KUKA KRL program: style1drop1opt1.src, style1drop1opt1.dat

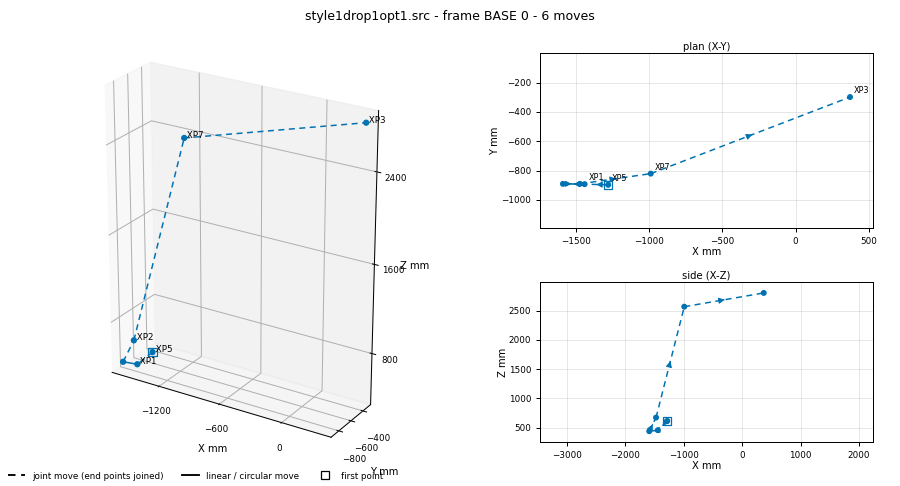
[picture p0: tool path of style1drop1opt1.src in frame BASE 0, 6 of 7 moves have a stored position in this frame; points joined in program order, loops and branches not executed]
--- style1drop1opt1.src ---
&ACCESS RVO1
&REL 222
&COMMENT 03-10-R1 DROP CONVEYOR
&PARAM EDITMASK = *
&PARAM DISKPATH = KRC:\R1\Program\StyleDrops\Options
DEF Style1Drop1Opt1( )
   ;FOLD INI
      ;FOLD BASISTECH INI
         GLOBAL INTERRUPT DECL 3 WHEN $STOPMESS==TRUE DO IR_STOPM ( )
         INTERRUPT ON 3
         BAS (#INITMOV,0 )
      ;ENDFOLD (BASISTECH INI)
      ;FOLD USER INI
         ;Make your modifications here

      ;ENDFOLD (USER INI)
   ;ENDFOLD (INI)
;********************************
; Gestamp Standards
; Line - BMW G65 (cell 03)
; Robot 03-10-R1 (BMW-03-10-R1-MH1)
; Application - DROP THE GOOD PART AT DROPOFF 1 (CONVEYOR)
;********************************
; CALLED BY Style1Opt1 WHEN BOTH NUT CHECKS PASSED. PLACES THE PART AT AtDrop3, OPENS
; GRIPPER 1, WAITS FOR THE GRIPPER EMPTY, LEAVES AND RETURNS HOME.
;NOTE: THE PART IN THE GRIPPER IS NOT CONFIRMED BEFORE OPENING (F40)
;DROPOFF 1 REQUEST - AC_DropOffCheck(1): WAIT SIGNAL $IN[75] di075DropOffMachine1 ON
;(WAITING MESSAGE, NO TIMEOUT), THEN SIGNALS $OUT[75] do075DropOffClear1 OFF,
;$OUT[25] do025DropClearTooling OFF
;WARNING: HIDDEN AC_CmdParam=2 - CONFIRMING THIS FORM REGENERATES AC_DropOffCheck(2) (F21)
;FOLD DropOff[1] Request
;FOLD ;%{h}
;Params IlfProvider=ac_zoneilf; AC_CmdZones=DropOff; AC_CmdParam=2; AC_ZoneRepo=False; AC_Blending=False
;ENDFOLD
AC_DropOffCheck (1)
;ENDFOLD

;APPROACH DROPOFF 1 - P5, P1, AtDrop3 (DROP POSITION)
;FOLD PTP P5 CONT Vel=100 % PDAT10 Tool[1]:TOOL 1 Base[0];%{PE}%R 8.3.43,%MKUKATPBASIS,%CMOVE,%VPTP,%P 1:PTP, 2:P5, 3:C_DIS, 5:100, 7:PDAT10
$BWDSTART=FALSE
PDAT_ACT=PPDAT10
FDAT_ACT=FP5
BAS(#PTP_PARAMS,100)
PTP XP5 C_DIS
;ENDFOLD
;FOLD PTP P1 Vel=100 % PDAT1 Tool[1]:TOOL 1 Base[0];%{PE}%R 8.3.43,%MKUKATPBASIS,%CMOVE,%VPTP,%P 1:PTP, 2:P1, 3:, 5:100, 7:PDAT1
$BWDSTART=FALSE
PDAT_ACT=PPDAT1
FDAT_ACT=FP1
BAS(#PTP_PARAMS,100)
PTP XP1
;ENDFOLD
;FOLD LIN AtDrop3 Vel=2 m/s CPDAT1 Tool[1]:TOOL 1 Base[0];%{PE}%R 8.3.43,%MKUKATPBASIS,%CMOVE,%VLIN,%P 1:LIN, 2:AtDrop3, 3:, 5:2, 7:CPDAT1
$BWDSTART=FALSE
LDAT_ACT=LCPDAT1
FDAT_ACT=FAtDrop3
BAS(#CP_PARAMS,2)
LIN XAtDrop3
;ENDFOLD

;GRIPPER 1 OPEN - SIGNALS $OUT[249] do249Group1Home ON, $OUT[250] do250Group1Work OFF, WAIT 0.2 S,
;THEN CHECK $IN[257] di257Cylinder1Home ON, $IN[258] di258Cylinder1Work OFF (STRATEGY 1)
;WARNING: THE HIDDEN FORM PARAMETERS SAY setgripper=4;setstate=2 - OPENING AND CONFIRMING THIS
;  FORM REGENERATES GRPg_SetStateAndCheck(4, 2, ...), AN INACTIVE GRIPPER: NOTHING OPENS (F31)
   ;FOLD Gripper SET [1]Gripper1 State=[1]OPEN Wait 0.2[s] Check with Strategy 1 ;%{PE}
      ;FOLD Parameters Parameters ;%{h}
         ;Params IlfProvider=GripperTech.GripperSet;setgripper=4;setstate=2;setcont=nocont;waittime=0.2;errorstrategy=1
      ;ENDFOLD
      GRPg_SetStateAndCheck(1, 1, 0.2, 1)
   ;ENDFOLD
;CHECK GRIPPER 1 OPEN AGAIN (REPEATS THE CHECK ABOVE)
;FOLD Gripper CHECK [1]Gripper 1 State=[1]OPEN with Strategy 1 ;%{PE}
;FOLD Parameters Parameters ;%{h}
;Params IlfProvider=GripperTech.GripperCheck;setgripper=1;setstate=1;setcont=nocont;checkstrategy=1
;ENDFOLD
GRPg_Check(1, 1, FALSE, 1)
;ENDFOLD
;WAIT GRIPPER EMPTY - SIGNALS $IN[253] di253PartPresent1 OFF, $IN[254] di254PartPresent2 OFF (NO TIMEOUT)
;FOLD WAIT FOR ( NOT IN 253 'di253PartPresent1' ) AND ( NOT IN 254 'di254PartPresent2' );%{PE}%R 8.3.43,%MKUKATPBASIS,%CEXT_WAIT_FOR,%VEXT_WAIT_FOR,%P 2:, 4:NOT, 5:$IN, 6:253, 7:di253PartPresent1, 9:AND, 10:, 12:NOT, 13:$IN, 14:254, 15:di254PartPresent2, 17:
WAIT FOR  (  NOT $IN[253] ) AND (  NOT $IN[254] )
;ENDFOLD
;PART NOT IN GRIPPER - SIGNAL $OUT[18] do018Part1InGripper OFF
;FOLD OUT 18 'do018PartInGripper1' State=FALSE ;%{PE}%R 8.3.43,%MKUKATPBASIS,%COUT,%VOUTX,%P 2:18, 3:do018PartInGripper1, 5:FALSE, 6:
$OUT[18]=FALSE
;ENDFOLD

;LEAVE DROPOFF 1 - P2, P7, P3
;FOLD PTP P2 CONT Vel=100 % PDAT7 Tool[1]:TOOL 1 Base[0];%{PE}%R 8.3.43,%MKUKATPBASIS,%CMOVE,%VPTP,%P 1:PTP, 2:P2, 3:C_DIS, 5:100, 7:PDAT7
$BWDSTART=FALSE
PDAT_ACT=PPDAT7
FDAT_ACT=FP2
BAS(#PTP_PARAMS,100)
PTP XP2 C_DIS
;ENDFOLD

;FOLD PTP P7 CONT Vel=100 % PDAT13 Tool[1]:TOOL 1 Base[0];%{PE}%R 8.3.43,%MKUKATPBASIS,%CMOVE,%VPTP,%P 1:PTP, 2:P7, 3:C_DIS, 5:100, 7:PDAT13
$BWDSTART=FALSE
PDAT_ACT=PPDAT13
FDAT_ACT=FP7
BAS(#PTP_PARAMS,100)
PTP XP7 C_DIS
;ENDFOLD
;FOLD PTP P3 Vel=100 % PDAT2 Tool[1]:TOOL 1 Base[0];%{PE}%R 8.3.43,%MKUKATPBASIS,%CMOVE,%VPTP,%P 1:PTP, 2:P3, 3:, 5:100, 7:PDAT2
$BWDSTART=FALSE
PDAT_ACT=PPDAT2
FDAT_ACT=FP3
BAS(#PTP_PARAMS,100)
PTP XP3
;ENDFOLD

;DROPOFF 1 CLEAR - AC_DropOff(1,TRUE): SIGNAL $OUT[75] do075DropOffClear1 ON
;WARNING: HIDDEN AC_CmdParam=2 - CONFIRMING THIS FORM REGENERATES AC_DropOff(2,TRUE) (F21)
;FOLD DropOff[1] Reset
;FOLD ;%{h}
;Params IlfProvider=ac_zoneilf; AC_CmdZones=DropOff; AC_CmdParam=2; AC_ZoneRepo=True; AC_Blending=False
;ENDFOLD
AC_DropOff (1,True)
;ENDFOLD

;PTP HOME (XHOME)
;FOLD PTP HOME Vel=100 % PDAT11;%{PE}%R 8.3.43,%MKUKATPBASIS,%CMOVE,%VPTP,%P 1:PTP, 2:HOME, 3:, 5:100, 7:PDAT11
$BWDSTART=FALSE
PDAT_ACT=PPDAT11
FDAT_ACT=FHOME
BAS(#PTP_PARAMS,100)
$H_POS=XHOME
PTP XHOME
;ENDFOLD

END

--- style1drop1opt1.dat ---
&ACCESS RVO1
&REL 222
&COMMENT GE4_Conveyor
&PARAM EDITMASK = *
&PARAM DISKPATH = KRC:\R1\Program\StyleDrops\Options
DEFDAT  style1drop1opt1
;FOLD EXTERNAL DECLARATIONS;%{PE}%MKUKATPBASIS,%CEXT,%VCOMMON,%P
EXT  BAS (BAS_COMMAND  :IN,REAL  :IN )
DECL INT SUCCESS
;ENDFOLD (BASISTECH EXT)
;FOLD USER EXT;%{E}%MKUKATPUSER,%CEXT,%VEXT,%P
;Make here your modifications

;ENDFOLD (USER EXT)
;ENDFOLD (EXTERNAL DECLARATIONS)
DECL BASIS_SUGG_T LAST_BASIS={POINT1[] "P10                     ",POINT2[] "P10                     ",CP_PARAMS[] "CPDAT0                  ",PTP_PARAMS[] "PDAT6                   ",CONT[] "                        ",CP_VEL[] "2                       ",PTP_VEL[] "100                     ",SYNC_PARAMS[] "SYNCDAT                 ",SPL_NAME[] "S0                      ",A_PARAMS[] "ADAT0                   "}
DECL E6POS XATDROP3={X -1587.76917,Y -890.400757,Z 439.605072,A 177.082932,B 4.31955290,C -0.298484027,S 2,T 2,E1 0.0,E2 0.0,E3 0.0,E4 0.0,E5 0.0,E6 0.0}
DECL FDAT FAtDrop3={TOOL_NO 1,BASE_NO 0,IPO_FRAME #BASE,POINT2[] " ",TQ_STATE FALSE}
DECL MODULEPARAM_T LAST_TP_PARAMS={PARAMS[] "AC_CmdZones=DropOff; AC_CmdParam=2; AC_ZoneRepo=True; AC_UseState=True; AC_Blending=False                               "}
DECL E6POS XP2={X -1471.65808,Y -890.400757,Z 672.790649,A 177.082932,B 4.31955290,C -0.298484206,S 2,T 2,E1 0.0,E2 0.0,E3 0.0,E4 0.0,E5 0.0,E6 0.0}
DECL FDAT FP2={TOOL_NO 1,BASE_NO 0,IPO_FRAME #BASE,POINT2[] " ",TQ_STATE FALSE}
DECL PDAT PPDAT7={VEL 100.000,ACC 100.000,APO_DIST 500.000,APO_MODE #CDIS,GEAR_JERK 50.0000,EXAX_IGN 0}
DECL E6POS XP5={X -1279.37976,Y -897.098,Z 616.329468,A 176.629059,B 21.7134552,C -1.31570351,S 2,T 2,E1 0.0,E2 0.0,E3 0.0,E4 0.0,E5 0.0,E6 0.0}
DECL FDAT FP5={TOOL_NO 1,BASE_NO 0,IPO_FRAME #BASE,POINT2[] " ",TQ_STATE FALSE}
DECL PDAT PPDAT10={VEL 100.000,ACC 100.000,APO_DIST 500.000,APO_MODE #CDIS,GEAR_JERK 50.0000,EXAX_IGN 0}
DECL PDAT PPDAT11={VEL 100.000,ACC 100.000,APO_DIST 100.000,GEAR_JERK 50.0000,EXAX_IGN 0}
DECL PDAT PPDAT13={VEL 100.000,ACC 100.000,APO_DIST 500.000,APO_MODE #CDIS,GEAR_JERK 50.0000,EXAX_IGN 0}
DECL E6POS XP7={X -988.705139,Y -820.766479,Z 2569.14844,A 137.545090,B -48.9822197,C 56.5858917,S 2,T 2,E1 0.0,E2 0.0,E3 0.0,E4 0.0,E5 0.0,E6 0.0}
DECL FDAT FP7={TOOL_NO 1,BASE_NO 0,IPO_FRAME #BASE,POINT2[] " ",TQ_STATE FALSE}
DECL E6POS XP1={X -1440.21106,Y -892.543274,Z 457.022766,A 177.090073,B 1.60787833,C -0.160304546,S 2,T 2,E1 0.0,E2 0.0,E3 0.0,E4 0.0,E5 0.0,E6 0.0}
DECL FDAT FP1={TOOL_NO 1,BASE_NO 0,IPO_FRAME #BASE,POINT2[] " ",TQ_STATE FALSE}
DECL PDAT PPDAT1={VEL 100.000,ACC 100.000,APO_DIST 100.000,APO_MODE #CDIS,GEAR_JERK 50.0000,EXAX_IGN 0}
DECL E6POS XP3={X 370.852905,Y -298.257416,Z 2804.38916,A -147.361786,B -35.6047363,C 79.4075775,S 2,T 2,E1 0.0,E2 0.0,E3 0.0,E4 0.0,E5 0.0,E6 0.0}
DECL FDAT FP3={TOOL_NO 1,BASE_NO 0,IPO_FRAME #BASE,POINT2[] " ",TQ_STATE FALSE}
DECL PDAT PPDAT2={VEL 100.000,ACC 100.000,APO_DIST 100.000,APO_MODE #CDIS,GEAR_JERK 50.0000,EXAX_IGN 0}
DECL LDAT LCPDAT1={VEL 2.00000,ACC 100.000,APO_DIST 100.000,APO_FAC 50.0000,AXIS_VEL 100.000,AXIS_ACC 100.000,ORI_TYP #VAR,CIRC_TYP #BASE,JERK_FAC 50.0000,GEAR_JERK 50.0000,EXAX_IGN 0}
ENDDAT
